# EPICS IOC start-up script: calcApp/iocsh/userCalc_extra.iocsh
# ### userCalc.iocsh ###

#- ###################################################
#- PREFIX         - IOC Prefix
#- CALC           - Location of Calc module
#- N              - Additional calcs index (Ex: N=1 creates calcs 10-19)
#- ARRAY_SIZE     - Optional: Size of userArrayCalc array
#-                  Default:  8000
#- ###################################################

#- ## Stuff for user programming ###
dbLoadRecords("$(CALC)/db/userCalcs10more.db","P=$(PREFIX),N10=$(N)0,N1=$(N)1,N2=$(N)2,N3=$(N)3,N4=$(N)4,N5=$(N)5,N6=$(N)6,N7=$(N)7,N8=$(N)8,N9=$(N)9")
dbLoadRecords("$(CALC)/db/userCalcOuts10more.db","P=$(PREFIX),N10=$(N)0,N1=$(N)1,N2=$(N)2,N3=$(N)3,N4=$(N)4,N5=$(N)5,N6=$(N)6,N7=$(N)7,N8=$(N)8,N9=$(N)9")
dbLoadRecords("$(CALC)/db/userStringCalcs10more.db","P=$(PREFIX),N10=$(N)0,N1=$(N)1,N2=$(N)2,N3=$(N)3,N4=$(N)4,N5=$(N)5,N6=$(N)6,N7=$(N)7,N8=$(N)8,N9=$(N)9")
dbLoadRecords("$(CALC)/db/userArrayCalcs10more.db","P=$(PREFIX),N10=$(N)0,N1=$(N)1,N2=$(N)2,N3=$(N)3,N4=$(N)4,N5=$(N)5,N6=$(N)6,N7=$(N)7,N8=$(N)8,N9=$(N)9,N=$(ARRAY_SIZE=8000)")
dbLoadRecords("$(CALC)/db/userTransforms10more.db","P=$(PREFIX),N10=$(N)0,N1=$(N)1,N2=$(N)2,N3=$(N)3,N4=$(N)4,N5=$(N)5,N6=$(N)6,N7=$(N)7,N8=$(N)8,N9=$(N)9")
dbLoadRecords("$(CALC)/db/userAve10more.db","P=$(PREFIX),N10=$(N)0,N1=$(N)1,N2=$(N)2,N3=$(N)3,N4=$(N)4,N5=$(N)5,N6=$(N)6,N7=$(N)7,N8=$(N)8,N9=$(N)9")
